# B&R Automation Studio project JOB_NUMBER (part 8)

### Device.var
```iecst
VAR
	Device : ARRAY[0..MAX_DEVICES] OF Device_typ := [(RequestRelease:=0,ReadyToRecieve:=0,Recieved:=0),221(0)];
END_VAR
VAR CONSTANT
	DEVICE_RELEASE_ID : UINT := 999; (**Value that is set in RequestRelease, when the destination is not required*)
	DEVICE_RELEASE_EMPTY : UINT := 998; (**Value that is set in RequestRelease, when the empty bag is required*)
	DEVICE_RECIEVE_WAIT : UINT := 997; (**Special ID to show a device is able to recieve but will not explicitly enable any sequence*)
END_VAR
```

### Device_IDS.var
```iecst
VAR CONSTANT
	MAX_DEVICES : UINT := 240;
END_VAR
(**Device ID constants*)
VAR CONSTANT
	DEVICE_LINE : ARRAY[0..99] OF UINT := [0,1,2,3,4,5,6,7,8,9,10,11,12,13,14,15,16,17,18,19,20,21,22,23,24,25,26,27,28,29,30,31,32,33,34,35,36,37,38,39,40,41,42,43,44,45,46,47,48,49,50,51,52,53,54,55,56,57,58,59,60,61,62,63,64,65,66,67,68,69,70,71,72,73,74,75,76,77,78,79,80,81,82,83,84,85,86,87,88,89,90,91,92,93,94,95,96,97,98,99]; (*Lines ID 1-99*)
	DEVICE_BSN : ARRAY[0..5] OF UINT := [0,101,102,103,104,105]; (*Bag Stacker Ongoing 101 - 105*)
	DEVICE_BSF : ARRAY[0..5] OF UINT := [0,106,107,108,109,110]; (*Bag Stacker Offgoing 106 - 110*)
	DEVICE_DC : ARRAY[0..10] OF UINT := [0,111,112,113,114,115,116,117,118,119,120]; (*Dischargers 111-120*)
	DEVICE_IC : ARRAY[0..10] OF UINT := [0,121,122,123,124,125,126,127,128,129,130]; (*Electric Inclines 121 - 130*)
	DEVICE_VC : ARRAY[0..10] OF UINT := [0,131,132,133,134,135,136,137,138,139,140]; (*VCs & Hoists 131 - 140*)
	DEVICE_TB : ARRAY[0..5] OF UINT := [0,141,142,143,144,145]; (*Transfer Belts 141 - 145*)
	DEVICE_PN : ARRAY[0..2] OF UINT := [0,146,147]; (*Ongoing Points 146 - 147*)
	DEVICE_PF : ARRAY[0..2] OF UINT := [0,148,149]; (*Points 148 - 149*)
	DEVICE_RPN : ARRAY[0..5] OF UINT := [0,151,152,153,154,155]; (*Rotary Ongoing 151-155*)
	DEVICE_RPF : ARRAY[0..5] OF UINT := [0,156,157,158,159,160]; (*Rotary Offgoing 156-160*)
	DEVICE_PC : ARRAY[0..10] OF UINT := [0,171,172,173,174,175,176,177,178,179,180]; (*Pneumatic VC 171-180*)
	DEVICE_PI : ARRAY[0..10] OF UINT := [0,181,182,183,184,185,186,187,188,189,190]; (*Pneumatic IC 181-190*)
	DEVICE_LU : ARRAY[0..10] OF UINT := [0,191,192,193,194,195,196,197,198,199,200]; (*Loading Units 191-200*)
	DEVICE_TRN : ARRAY[0..10] OF UINT := [0,201,202,203,204,205,206,207,208,209,210]; (*Twin Rail ongoing 201-205*)
	DEVICE_TRF : ARRAY[0..10] OF UINT := [0,211,212,213,214,215,216,217,218,219,220]; (*Twin Rail Offgoing 206-210*)
	DEVICE_POINT : ARRAY[0..20] OF UINT := [0,221,222,223,224,225,226,227,228,229,230,231,232,233,234,235,236,237,238,239,240]; (*Points 151 - 170*)
END_VAR
```

### Types.typ - Exported data types
```iecst
TYPE
	http_comm_typ : 	STRUCT
		Command : http_Cmd_typ; (**Set the values to pass into the http comm driver,*)
		Status : HTTP_Status_enum; (**Status of the http comm driver.*)
		LastError : STRING[60]; (**String to describe the last error*)
		lastResponse : httpResponseHeader_t;
		Overwrite : http_overwrite_t;
		ReplyCode : UINT; (**The response code *)
	END_STRUCT;
	http_Cmd_typ : 	STRUCT
		Method : UINT; (*Set the http cmd type.. POST,GET,PUT,DELETE*)
		Cmd_URL : dataPointer_typ; (*The string data appended to the URL - Use with GET and DELETE *)
		Body_Data : dataPointer_typ; (*Data to send in the body of the message - USE with POST and PUT*)
		ResponseData : dataPointer_typ; (*Data address of where to set the http response data*)
	END_STRUCT;
	dataPointer_typ : 	STRUCT
		Adr : UDINT;
		Size : UDINT;
	END_STRUCT;
	HTTP_Status_enum :
		(
		HTTP_COMM_STATUS_DISABLED,
		HTTP_COMM_STATUS_ACTIVE_WAIT_BUF,
		HTTP_COMM_STATUS_IN_BUFFER,
		HTTP_COMM_STATUS_IN_PROCESS,
		HTTP_COMM_STATUS_COMPLETE,
		HTTP_COMM_STATUS_ERROR
		);
	httpConfig_typ : 	STRUCT
		Host : STRING[20];
		Port : UINT;
	END_STRUCT;
	http_overwrite_t : 	STRUCT
		Host : BOOL; (**Set this to overwrite the host name and Port*)
		RequestHeader : BOOL; (**Set this to overwrite the Request Header*)
		Host_Config : httpConfig_typ; (**This data will overwrite the default host config*)
		RequestHeader_Data : httpRequestHeader_t; (**This data will overwrite the default request header.*)
	END_STRUCT;
END_TYPE
```

### Program Logical/Bag/http_Lib/httpServer (IEC, version 2.00.7) - *Listen for http requests

#### Variables.var - Local variables
```iecst
VAR
	httpServer : httpService;
	sendResponse : BOOL;
	abortResponse : BOOL;
	URI : STRING[500];
	requestHeader : httpRequestHeader_t;
	requestData : STRING[10000];
	responseHeader : httpResponseHeader_t;
	responseData : STRING[10000];
	Statistics : httpStatistics_t;
	serviceName : STRING[50];
	getParameterName : httpGetParameter;
END_VAR
VAR CONSTANT
	STRING_DOLLAR : STRING[1] := '&';
END_VAR
VAR
	activeFunction : UINT;
	mis : UDINT;
	bagIndex : UDINT;
	dst : USINT;
	error : INT;
	api : UINT;
	errorResponse : BOOL;
	overRideData : overRide_typ;
	ton_httpTimeOut : TON_10ms;
	recv : R_TRIG;
	wait : F_TRIG;
	cat : UDINT;
	cus : UDINT;
	bag : REFERENCE TO Bag_typ;
	prg : USINT;
	found : USINT;
	recieved : BOOL;
END_VAR
VAR CONSTANT
	BLANK_RESPONSE_HEADER : httpResponseHeader_t := (0);
END_VAR
VAR
	requestArriveTime : DATE_AND_TIME;
	debugCount : UDINT;
	index : UDINT;
	belt : USINT;
	velocity : INT;
(*	PartLoad : ARRAY[0..MAX_DISPLAYS] OF BOOL;*)
	direction : USINT;
	command : USINT;
END_VAR
```

#### Main.st - Init, cyclic, exit code
```iecst
//V2.00.1 -- TR. First release using version numbering
//V2.00.2 -- TR. Remove old http server functions FOR ABB settings as vars have been removed
//		  -- FIX: 200 OK could be returned in error
//V2.00.3 -- ADD: Load new configuration file command
//V2.00.4 -- REMOVE: Clear up old API Calls
//V2.00.5 -- Add Discharger Displays
//V2.00.6 -- ADD Part load and ABB Manual Controls (NEEDS ABB DRIVER 3.00.2)
//V2.00.7 -- ADD more functionality to ABB Manual Controls (Command and Direction) -- Also startup UDP Data connection
PROGRAM _INIT
	serviceName := 'supertrackPLC.api';
	httpServer.pServiceName := ADR(serviceName);
	httpServer.pUri := ADR(URI);
	httpServer.uriSize := SIZEOF(URI);
	httpServer.pRequestHeader := ADR(requestHeader);
	httpServer.pRequestData := ADR(requestData);
	httpServer.requestDataSize := SIZEOF(requestData);
	httpServer.pResponseHeader := ADR(responseHeader);
	httpServer.pResponseData := ADR(responseData);

	httpServer.pStatistics := ADR(Statistics);

	httpServer.option := httpOPTION_HTTP_11 + httpOPTION_SERVICE_TYPE_ROOT; //HTTP 1.1
	httpServer.enable := 0;

END_PROGRAM

PROGRAM _CYCLIC

	_httpServer;

	wait(CLK := (httpServer.phase = httpPHASE_SENDING));
	recv(CLK := (httpServer.phase = httpPHASE_RECEIVED));
	IF wait.Q THEN
		memset(ADR(responseData),0,SIZEOF(responseData));//Clear responseData
	END_IF;

	IF EDGEPOS(recieved) THEN
		requestArriveTime := CurrentTimestamp; // Get time stamp when the request arrives.
	END_IF;

	IF recieved THEN//recv.Q THEN
		//Get the API!
		api := FindAPI(URI,serviceName);

		CASE api OF

			API_UNKNOWN:
				errorResponse := 1;
				overRideData.responseHeader.status := '501 Not Implemented';
				responseData := 'Unknown API';
				httpServer.responseDataLen := LEN(responseData);

			API_MAINTENANCE_CONFIRM_REENTRY:
				sendResponse := 1;

			API_ST_FUNCTIONS://Legacy function => ?function=xxx
				_apiFunctions;

			API_CONFIG_LOAD_NEW: // Request to load new configuration.
				IF (Configuration.Interface.Status.LastLoaded >= requestArriveTime)  THEN // Send 200 OK when we see that the configuration is newer than the previous
					sendResponse := 1;
				ELSIF Configuration.Interface.Status.Error THEN
					errorResponse := 1;
					overRideData.responseHeader.status := '500 Internal Server Error';
					responseData := 'Failed to load file';
					httpServer.responseDataLen := LEN(responseData);
				ELSIF NOT Configuration.Interface.Cmd.Load AND (Configuration.Interface.Status.LastLoaded < requestArriveTime) THEN
					Configuration.Interface.Cmd.Load := 1;
					debugCount := debugCount + 1;
				END_IF;

			API_DISCHARGER_SUBMIT:

				getParameterName.searchString := requestData;
				getParameterName.searchOffset := 0;
				getParameterName.searchEndProperty := STRING_DOLLAR;
				//Find the first part of the array in JSON
				getParameterName.searchPropertyName := 'playId":"';
				getParameterName.searchEndProperty := '",';
				getParameterName();
				IF (getParameterName.status = ERR_OK) THEN
					index := DINT_TO_UDINT(atoi(ADR(getParameterName.outputValue)));
					IF (index <= MAX_DISPLAYS) THEN
						DischargerDisplaySubmit[index] := 1;
					END_IF;
					sendResponse := 1;
				ELSE
					errorResponse := 1;
					overRideData.responseHeader.status := '404 Not Found';
					responseData := 'Unknown display';
					httpServer.responseDataLen := LEN(responseData);
				END_IF;

			API_ABB_MANUAL_CMD:
				_abbManual;

			API_DATA_ENTRY_PARTLOAD:
				getParameterName.searchString := requestData;
				getParameterName.searchOffset := 0;
				getParameterName.searchEndProperty := STRING_DOLLAR;
				//Find the first part of the array in JSON
				getParameterName.searchPropertyName := 'playId":';
				getParameterName.searchEndProperty := '}';
				getParameterName();
				IF (getParameterName.status = ERR_OK) THEN
					index := DINT_TO_UDINT(atoi(ADR(getParameterName.outputValue)));
					IF (index <= MAX_DISPLAYS) THEN
						PartLoad[index] := 1;
					END_IF;
					sendResponse := 1;
				ELSE
					errorResponse := 1;
					overRideData.responseHeader.status := '404 Not Found';
					responseData := 'Unknown display';
					httpServer.responseDataLen := LEN(responseData);
				END_IF;

			//			API_CUSTOM_BELT_CONFIG:
			//				_setBeltConfig;
			//				sendResponse := 1;
			//
			//			API_CUSTOM_VC_COMMAND:
			//				_vcCommand;
			//
			//			API_LOADING_DATA:
			//				_getLoadingData;

		END_CASE;
	ELSE
		api := 0;
		activeFunction := 0;
	END_IF;

END_PROGRAM

PROGRAM _EXIT
	//Disable the Server on Exit..
	httpServer.enable := 0;
	httpServer();
END_PROGRAM
```

### ContactronTrip.var
```iecst
VAR CONSTANT
	CONTACTRON_TRIP_MIN : USINT := 2#00000001; (*Overload current must be set in % in 15 increments*)
	CONTACTRON_TRIP_50_PERCENT : USINT := 2#00000111;
	CONTACTRON_TRIP_MAX : USINT := 2#00001111;
END_VAR
```

### IOLink.var
```iecst
VAR
	IO_Link : IO_Link_Type;
	Fuse_PB_Reset : ARRAY[0..2] OF BOOL;
	Fuse_PB_Lamp : ARRAY[0..2] OF BOOL;
END_VAR
```

### Program Logical/IOLink/IOLink_Driver (IEC)

#### Main.st - Init, cyclic, exit code
```iecst
(********************************************************************
 * COPYRIGHT --
 ********************************************************************
 * PROGRAM: IOLink
 * File: IOLink_Driver.st
 * Author: Stephen Healey
 * Created: Sept 05, 2018
 ********************************************************************
 * Implementation OF PROGRAM IOLink
 ********************************************************************)
//V1.00.1 First Release

//	Description
//IOLink task for controlling Contactron's and EasyB's
//Constants need to be set. MAX_CONTACTRON and MAX_EASYB should match the hardware
//IO needs to be mapped for the Contactron's in the X20DS438A
//EasyB's IO does not need mapping. The interface still needs enabling in the X20DS438A config

//-------------------------------------------------------------
//-----------------------------Init----------------------------
//-------------------------------------------------------------
//	1.	Configures IOLink physical device, adjust address as needed
//	2.	Resets the controller state, needs to start offset, not 0

//-------------------------------------------------------------
//-----------------------------Cyclic--------------------------
//-------------------------------------------------------------
//	1.	Calls contactron action only if MAX_CONTACTRON is greater than zero
//	2.	Calls easyB action only if MAX_EASYB is greater than zero
//	3.	Monitors tripped status of all the EasyB's and enables reseting

//Use the following charts when setting the trip currents for the IOLink devices

//Contactron 												EasyB
//Current Setting Chart							Current Setting Chart
//Bit 		Nominal current						Enum										USINT			Value
//3 2 1 0 [mA]																													[mA]
//				 3 A 9 A
//0 0 0 0 180 1500									TRIP_CURRENT_DEFAULT		0					N/A
//0 0 0 1 300 2000									TRIP_CURRENT_500mA			5					500
//0 0 1 0 440 2500									TRIP_CURRENT_1A					10				1000
//0 0 1 1 600 3000									TRIP_CURRENT_2A					20				2000
//0 1 0 0 680 3500									TRIP_CURRENT_3A					30				3000
//0 1 0 1 880 4000									TRIP_CURRENT_4A					40				4000
//0 1 1 0 1000 4500									TRIP_CURRENT_5A					50				5000
//0 1 1 1 1100 5000									TRIP_CURRENT_6A					60				6000
//1 0 0 0 1200 5500									TRIP_CURRENT_8A					80				8000
//1 0 0 1 1500 6000									TRIP_CURRENT_10A				100				10000
//1 0 1 0 1600 6500
//1 0 1 1 1900 7000
//1 1 0 0 2100 7500
//1 1 0 1 2400 8000
//1 1 1 0 2700 8500
//1 1 1 1 3000 9000

PROGRAM _INIT
	//Configuration

	//Reset state

	backUp.fileDevice := 'UserPart';
	backUp.filePath := 'FuseTripConfig';

	//Load from file on boot

	backUp.step := backUpOpen;

	FOR n := 1 TO MAX_CONTACTRON DO
		IO_Link.Contactron[n].Cmd.Direction			:= CONTACTRON_FORWARD;
		IO_Link.Contactron[n].Cmd.Reset_Automatic	:= 1;
	END_FOR;

END_PROGRAM

PROGRAM _CYCLIC
	//Call status
	IF IO_Link.Status THEN
	 _status;
	END_IF;

	//Call httpResponse conditionally
//	IF IO_Link.Load THEN
//		_backUpRead;
//		_encodeData;
//	END_IF;

	//Call httpRequest conditionally
//	IF IO_Link.Save THEN
//		_decodeData;
//		_backUpWrite;
//		_encodeData;
//	END_IF;

	//Call contactron action
	IF MAX_CONTACTRON > 0 THEN
		_Contactron;
	END_IF;

//	//Call easy b action
//	IF (MAX_EASYB > 0) AND (MAX_EASYB <= 40) THEN
//		_EasyB;
//
//		//Monitor Tripped status
//		IO_Link.EasyB.Tripped := FALSE;
//		FOR n:=1 TO MAX_EASYB DO
//			IF IO_Link.EasyB.EasyB_Array[n].Status.TripState = EASYB_TRIPPED THEN
//				IO_Link.EasyB.Tripped := TRUE;
//				EXIT;
//			END_IF;
//		END_FOR;
//		//Reset Tripped status
//		IF IO_Link.EasyB.Tripped AND IO_Link.EasyB.Reset THEN
//			FOR n:=1 TO MAX_EASYB DO
//				IF IO_Link.EasyB.EasyB_Array[n].Status.TripState = EASYB_TRIPPED THEN
//					IO_Link.EasyB.EasyB_Array[n].Cmd.Reset := TRUE;
//				END_IF;
//			END_FOR;
//			IO_Link.EasyB.Reset := FALSE;
//		END_IF;
//		IO_Link.EasyB.TrippedLamp := IO_Link.EasyB.Tripped AND Std.Clock1s;
//	END_IF;

END_PROGRAM
```

#### _Contactron.st
```iecst
ACTION _Contactron:
	//----------------------------------------------
	//-----------------Contactron-------------------
	//----------------------------------------------

	//Write control word
	FOR n:=1 TO MAX_CONTACTRON DO
		IO_Link.Contactron[n].Comms.Read.CurrentActual := IO_Link.Contactron[n].Comms.Read.Data[0];
		IO_Link.Contactron[n].Comms.Read.DeviceType := IO_Link.Contactron[n].Comms.Read.Data[1];
		IO_Link.Contactron[n].Comms.Read.ThermalPercentOfMax := IO_Link.Contactron[n].Comms.Read.Data[2];
		IO_Link.Contactron[n].Comms.Read.CurrentPercentOfMax := IO_Link.Contactron[n].Comms.Read.Data[3];
		IO_Link.Contactron[n].Comms.Read.CurrentStatus := IO_Link.Contactron[n].Comms.Read.Data[4];
		IO_Link.Contactron[n].Comms.Read.Diagnostics := IO_Link.Contactron[n].Comms.Read.Data[5];

		CASE IO_Link.Contactron[n].Cmd.Direction OF
			CONTACTRON_FORWARD:
				IO_Link.Contactron[n].Comms.Write.Control.0 := IO_Link.Contactron[n].Cmd.Run;
				IO_Link.Contactron[n].Comms.Write.Control.7 := IO_Link.Contactron[n].Cmd.Run;
				IO_Link.Contactron[n].Comms.Write.Control.1 := FALSE;
				IO_Link.Contactron[n].Comms.Write.Control.5 := FALSE;

			CONTACTRON_REVERSE:
				IO_Link.Contactron[n].Comms.Write.Control.0 := FALSE;
				IO_Link.Contactron[n].Comms.Write.Control.7 := FALSE;
				IO_Link.Contactron[n].Comms.Write.Control.1 := IO_Link.Contactron[n].Cmd.Run;
				IO_Link.Contactron[n].Comms.Write.Control.5 := IO_Link.Contactron[n].Cmd.Run;

			ELSE
				IO_Link.Contactron[n].Comms.Write.Control.0 := FALSE;
				IO_Link.Contactron[n].Comms.Write.Control.7 := FALSE;
				IO_Link.Contactron[n].Comms.Write.Control.1 := FALSE;
				IO_Link.Contactron[n].Comms.Write.Control.5 := FALSE;

		END_CASE;

		IO_Link.Contactron[n].Comms.Write.Control.2 := IO_Link.Contactron[n].Cmd.Reset_Manual;
		IO_Link.Contactron[n].Comms.Write.Control.3 := IO_Link.Contactron[n].Cmd.Reset_Automatic;
		IO_Link.Contactron[n].Comms.Write.Control.4 := FALSE; //NOT USED
		IO_Link.Contactron[n].Comms.Write.Control.6 := IO_Link.Contactron[n].Cmd.Stop;

		IF IO_Link.Contactron[n].Cmd.Current > 0 THEN //Write trip current level
			IO_Link.Contactron[n].Comms.Write.NominalCurrent := (IO_Link.Contactron[n].Cmd.Current OR CONTACTRON_WRITE_CURRENT);
		ELSE
			IO_Link.Contactron[n].Comms.Write.NominalCurrent := 0;
		END_IF;
		IF IO_Link.Contactron[n].Cmd.Current = (IO_Link.Contactron[n].Comms.Read.CurrentStatus AND CONTACTRON_CURRENT_STATUS) THEN
			IO_Link.Contactron[n].Cmd.Current := 0; //Reset trip current if cmd written
		END_IF;

		//Read status
		IO_Link.Contactron[n].Status.Error := IO_Link.Contactron[n].Comms.Read.Diagnostics.0;
		IO_Link.Contactron[n].Status.STO_Active := NOT IO_Link.Contactron[n].Comms.Read.Diagnostics.3;
		IO_Link.Contactron[n].Status.Device_Ok := IO_Link.Contactron[n].Comms.Read.Diagnostics.5;
		IO_Link.Contactron[n].Status.Overload_Warning := IO_Link.Contactron[n].Comms.Read.Diagnostics.6;
		IO_Link.Contactron[n].Status.MainsFailure := ((IO_Link.Contactron[n].Comms.Read.CurrentStatus AND CONTACTRON_TRIP_STATUS) = CONTACTRON_MAINS_LOSS);
		IO_Link.Contactron[n].Status.PhaseLoss := ((IO_Link.Contactron[n].Comms.Read.CurrentStatus AND CONTACTRON_TRIP_STATUS) = CONTACTRON_PHASE_LOSS);
		IO_Link.Contactron[n].Status.Current := IO_Link.Contactron[n].Comms.Read.CurrentActual * 0.01;
		IO_Link.Contactron[n].Status.DeviceType := IO_Link.Contactron[n].Comms.Read.DeviceType;

		IF 	(IO_Link.Contactron[n].Comms.Read.CurrentStatus = 0) THEN
			IO_Link.Contactron[n].Cmd.Current				:= CONTACTRON_TRIP_50_PERCENT;
		END_IF;

	END_FOR;
END_ACTION
```

### Program Logical/IOLink/FuseManagement (IEC, version 1.00.2)

#### Main.st - Init, cyclic, exit code
```iecst
//V1.00.0 -- First Release
//V1.00.1 -- Update so we monitor the status of the fuse and can send reset commands
//V1.00.2 -- Invert the fault lamp to a healthy lamp to stay consistent with hardwired devices

PROGRAM _INIT
Fuse[1].pDevice := ADR('SL1.IF1.ST11.IF1.ST8.IF1');//'SL1.IF1.ST2.IF1.ST7.IF1');
Fuse[2].pDevice := ADR('SL1.IF1.ST11.IF1.ST8.IF2');
Fuse[3].pDevice := ADR('SL1.IF1.ST11.IF1.ST8.IF3');
Fuse[4].pDevice := ADR('SL1.IF1.ST11.IF1.ST8.IF4');
Fuse[5].pDevice := ADR('SL1.IF1.ST21.IF1.ST8.IF1');
Fuse[6].pDevice := ADR('SL1.IF1.ST21.IF1.ST8.IF2');
Fuse[7].pDevice := ADR('SL1.IF1.ST21.IF1.ST8.IF3');
Fuse[8].pDevice := ADR('SL1.IF1.ST21.IF1.ST8.IF4');

FOR n := 1 TO MAX_FUSE_BANKS DO
	fuse ACCESS ADR(Fuse[n]);
	fuse.Write.MinVoltage := 1800;
	fuse.Write.MaxVoltage := 2800;
	FOR i := 1 TO MAX_FUSES DO
		fuse.Write.Channel[i].Status := EB_STATE_ON;
		fuse.Write.Channel[i].TripCurrent := 40;
	END_FOR;
	fuse.index := 90;
	fuse.readStatusOnly := 0;
	fuseTrippedAlarm[n] := 0;
END_FOR;

//alarm 	ACCESS ADR(Alarm[208]);
END_PROGRAM

PROGRAM _CYCLIC

IF EDGEPOS(X[1003].X04) THEN
	reset[0] := 1;
END_IF;
IF EDGEPOS(X[2003].X04) THEN
	reset[1] := 1;
END_IF;

fuseFault[0] := 0;
fuseFault[1] := 0;
//alarm.On	:= 0;
//alarm.Name	:= 0;

FOR n := 1 TO MAX_FUSE_BANKS DO
	fuse ACCESS ADR(Fuse[n]);
	read ACCESS ADR(fuse.IOLinkRead);
	write ACCESS ADR(fuse.IOLinkWrite);

	read.enable := 1;
	write.enable := 1;
	write.pDeviceName 	:= fuse.pDevice;
	read.pDeviceName 	:= fuse.pDevice;

	IF EDGEPOS(read.readLen > 0) THEN
		count := count + 1;
	END_IF;

	IF (read.errorCode > 0) THEN
		fuse.index := 10;
	END_IF;

	IF (n < 5) THEN
		plc := 0;
	ELSE
		plc := 1;
	END_IF;

	CASE fuse.index	OF
		0:

		32:	//Read Error Count
			read.datatype 		:= ioLinkTYPE_SINT;
			read.pData			:= ADR(fuse.Read.ErrorCount);
			read.dataLen		:= SIZEOF(fuse.Read.ErrorCount);
			read.index			:= fuse.index;
			read.subIndex		:= 0;
			read();
			IF read.status = ERR_OK THEN
				fuse.index := fuse.index + 1;
			ELSIF (read.status <> ERR_FUB_BUSY) AND (read.status <> ERR_FUB_ENABLE_FALSE)  THEN
				fuse.index := fuse.index + 1;
				//fuse.Read.ErrorCount := 0;
			END_IF;

		33://
			fuse.index := 36;

		36://Device Status	 R/O USINT
			read.datatype 		:= ioLinkTYPE_SINT;
			read.pData			:= ADR(fuse.Read.DeviceStatus);
			read.dataLen		:= SIZEOF(fuse.Read.DeviceStatus);
			read.index			:= fuse.index;
			read.subIndex		:= 0;
			read();
			IF read.status = ERR_OK THEN
				fuse.index := fuse.index + 1;
			ELSIF (read.status <> ERR_FUB_BUSY) AND (read.status <> ERR_FUB_ENABLE_FALSE)  THEN
				fuse.index := fuse.index + 1;
				//fuse.Read.ErrorCount := 0;
			END_IF;

		37:// Device Status	 R/O String
			read.datatype 		:= ioLinkTYPE_STRING;
			read.pData			:= ADR(fuse.Read.DeviceStatusString);
			read.dataLen		:= SIZEOF(fuse.Read.DeviceStatusString);
			read.index			:= fuse.index;
			read.subIndex		:= 0;
			read();
			IF read.status = ERR_OK THEN
				fuse.index := fuse.index + 1;
			ELSIF (read.status <> ERR_FUB_BUSY) AND (read.status <> ERR_FUB_ENABLE_FALSE)  THEN
				fuse.index := fuse.index + 1;
				//fuse.Read.ErrorCount := 0;
			END_IF;

		38:
			fuse.index := 80;

		80://
			IF (fuse.trip > 0) THEN
				command := UINT_TO_USINT((fuse.trip * 5) - 2); // <--RESET //((fuse.trip * 5) - 4); //<-- ON

				write.datatype 		:= ioLinkTYPE_USINT;
				write.pData			:= ADR(command);
				write.dataLen		:= SIZEOF(command);
				write.index			:= fuse.index;
				write.subIndex		:= 0;
				write();
				IF (write.status = ERR_OK) THEN
					fuse.index := fuse.index + 1;	;
				ELSIF (write.status <> ERR_FUB_BUSY) AND (write.status <> ERR_FUB_ENABLE_FALSE) THEN
					fuse.index := fuse.index + 1;
				END_IF;
			ELSE
				fuse.index := fuse.index + 1;
			END_IF;

		81://Gateway options ? R/W
			IF fuse.Write.AutoNodeAllocation_Off OR fuse.Write.AutoNodeAllocation_On  THEN
				//1 is automatic allocation off!
				//0 is on?
				IF fuse.Write.AutoNodeAllocation_Off THEN
					write.datatype 		:= ioLinkTYPE_RECORD;
					gatewayOption 		:= 1;
					write.subIndex		:= 1;
				ELSE
					write.datatype 		:= ioLinkTYPE_SINT;
					gatewayOption 		:= 0;
					write.subIndex		:= 0 ;
				END_IF;
				write.pData			:= ADR(gatewayOption);
				write.dataLen		:= 1;
				write.index			:= fuse.index;
				write();
				IF (write.status = ERR_OK) THEN
					fuse.index := fuse.index + 1;	;
					fuse.Write.AutoNodeAllocation_On := 0;
					fuse.Write.AutoNodeAllocation_Off := 0;
				ELSIF (write.status <> ERR_FUB_BUSY) AND (write.status <> ERR_FUB_ENABLE_FALSE) THEN
					fuse.index := fuse.index + 1;
					fuse.Write.AutoNodeAllocation_On := 0;
					fuse.Write.AutoNodeAllocation_Off := 0;
				END_IF;

			ELSE // Read if no write
				read.datatype 		:= ioLinkTYPE_SINT;
				read.pData			:= ADR(fuse.Read.GatewayOptions);
				read.dataLen		:= SIZEOF(fuse.Read.GatewayOptions);
				read.index			:= fuse.index;
				read.subIndex		:= 0;
				read();
				IF read.status = ERR_OK THEN
					fuse.index := fuse.index + 1;
				ELSIF (read.status <> ERR_FUB_BUSY) AND (read.status <> ERR_FUB_ENABLE_FALSE)  THEN
					fuse.index := fuse.index + 1;
				END_IF;
			END_IF;

		82://Set breaker 1 options to all
			fuse.index := 90;

		83:// Reset individual breaker.

		90://Input Voltage
			read.datatype 		:= ioLinkTYPE_INT;
			read.pData			:= ADR(fuse.Read.InputVoltage);
			read.dataLen		:= SIZEOF(fuse.Read.InputVoltage);
			read.index			:= fuse.index;
			read.subIndex		:= 0;
			read();
			IF read.status = ERR_OK THEN
				fuse.index := fuse.index + 1;
			ELSIF (read.status <> ERR_FUB_BUSY) AND (read.status <> ERR_FUB_ENABLE_FALSE)  THEN
				fuse.index := fuse.index + 1;
			END_IF;

		91://Number of Nodes
			read.datatype 		:= ioLinkTYPE_USINT;
			read.pData			:= ADR(fuse.Read.NoNodes);
			read.dataLen		:= SIZEOF(fuse.Read.NoNodes);
			read.index			:= fuse.index;
			read.subIndex		:= 0;
			read();
			IF read.status = ERR_OK THEN
				IF (fuse.Read.NoNodes > MAX_FUSES) THEN
					fuse.Read.NoNodes := MAX_FUSES;
				END_IF;
				fuse.index := fuse.index + 1;
			ELSIF (read.status <> ERR_FUB_BUSY) AND (read.status <> ERR_FUB_ENABLE_FALSE)  THEN
				fuse.Read.NoNodes := 0;
				fuse.index := fuse.index + 1;
			END_IF;

		92://
			fuse.index := 100;

		100:// Max Voltage
			IF (fuse.Write.MaxVoltage > 0) THEN

				write.datatype 		:= ioLinkTYPE_INT;
				write.pData			:= ADR(fuse.Write.MaxVoltage);
				write.dataLen		:= SIZEOF(fuse.Write.MaxVoltage);
				write.index			:= fuse.index;
				write.subIndex		:= 0;
				write();
				IF (write.status = ERR_OK) THEN
					fuse.index := fuse.index + 1;
					fuse.Read.MaxVoltage := fuse.Write.MaxVoltage;
					fuse.Write.MaxVoltage := 0;
				ELSIF (write.status <> ERR_FUB_BUSY) AND (write.status <> ERR_FUB_ENABLE_FALSE) THEN
					fuse.index := fuse.index + 1;
					fuse.Write.MaxVoltage := 0;
				END_IF;
			ELSE // Read if no write

				read.datatype 		:= ioLinkTYPE_INT;
				read.pData			:= ADR(fuse.Read.MaxVoltage);
				read.dataLen		:= SIZEOF(fuse.Read.MaxVoltage);
				read.index			:= fuse.index;
				read.subIndex		:= 0;
				read();
				IF read.status = ERR_OK THEN
					fuse.index := fuse.index + 1;
				ELSIF (read.status <> ERR_FUB_BUSY) AND (read.status <> ERR_FUB_ENABLE_FALSE)  THEN
					fuse.index := fuse.index + 1;
					fuse.Read.MaxVoltage := 0;
				END_IF;
			END_IF;

		101://MinVoltage
			IF (fuse.Write.MinVoltage > 0) THEN
				write.datatype 		:= ioLinkTYPE_INT;
				write.pData			:= ADR(fuse.Write.MinVoltage);
				write.dataLen		:= SIZEOF(fuse.Write.MinVoltage);
				write.index			:= fuse.index;
				write.subIndex		:= 0;
				write();
				IF (write.status = ERR_OK) THEN
					fuse.index := fuse.index + 1;
					fuse.Read.MinVoltage :=	fuse.Write.MinVoltage;
					fuse.Write.MinVoltage := 0;
				ELSIF (write.status <> ERR_FUB_BUSY) AND (write.status <> ERR_FUB_ENABLE_FALSE) THEN
					fuse.index := fuse.index + 1;
					fuse.Write.MinVoltage := 0;
				END_IF;
			ELSE // Read if no write

				read.datatype 		:= ioLinkTYPE_INT;
				read.pData			:= ADR(fuse.Read.MinVoltage);
				read.dataLen		:= SIZEOF(fuse.Read.MinVoltage);
				read.index			:= fuse.index;
				read.subIndex		:= 0;
				read();
				IF read.status = ERR_OK THEN
					fuse.index := fuse.index + 1;
				ELSIF (read.status <> ERR_FUB_BUSY) AND (read.status <> ERR_FUB_ENABLE_FALSE)  THEN
					fuse.index := fuse.index + 1;
					fuse.Read.MinVoltage := 0;
				END_IF;
			END_IF;

		102:// Enable Events R/W
			IF (fuse.Write.EnableEvents > 0) THEN
				write.datatype 		:= ioLinkTYPE_SINT;
				write.pData			:= ADR(fuse.Write.EnableEvents);
				write.dataLen		:= SIZEOF(fuse.Write.EnableEvents);
				write.index			:= fuse.index;
				write.subIndex		:= 0;
				write();
				IF (write.status = ERR_OK) THEN
					fuse.index := fuse.index + 1;
					fuse.Write.EnableEvents := 0;
				ELSIF (write.status <> ERR_FUB_BUSY) AND (write.status <> ERR_FUB_ENABLE_FALSE) THEN
					fuse.index := fuse.index + 1;
					fuse.Write.EnableEvents := 0;
				END_IF;
			ELSE // Read if no write

				read.datatype 		:= ioLinkTYPE_SINT;
				read.pData			:= ADR(fuse.Read.EnableEvents);
				read.dataLen		:= SIZEOF(fuse.Read.EnableEvents);
				read.index			:= fuse.index;
				read.subIndex		:= 0;
				read();
				IF read.status = ERR_OK THEN
					fuse.index := fuse.index + 1;
				ELSIF (read.status <> ERR_FUB_BUSY) AND (read.status <> ERR_FUB_ENABLE_FALSE)  THEN
					fuse.index := fuse.index + 1;
					fuse.Read.EnableEvents := 0;
				END_IF;
			END_IF;

		103:
			fuse.index := 201;

		201..240://Read Only Trip Counter
			index := (fuse.index - 200);
			read.datatype 		:= ioLinkTYPE_SINT;
			read.pData			:= ADR(fuse.Read.Channel[index].TripCount);
			read.dataLen		:= SIZEOF(fuse.Read.Channel[index].TripCount);
			read.index			:= fuse.index;
			read.subIndex		:= 0;
			read();
			IF read.status = ERR_OK THEN
				fuse.index := fuse.index + 1;
			ELSIF (read.status <> ERR_FUB_BUSY) AND (read.status <> ERR_FUB_ENABLE_FALSE)  THEN
				fuse.index := fuse.index + 1;
				//fuse.Read.Channel[index].TripCount := 0;
			END_IF;

		241:
			fuse.index := 301;

		301..340://Read only Actaul Current
			index := (fuse.index - 300);
			read.datatype 		:= ioLinkTYPE_INT;
			read.pData			:= ADR(fuse.Read.Channel[index].ActCurrent);
			read.dataLen		:= SIZEOF(fuse.Read.Channel[index].ActCurrent);
			read.index			:= fuse.index;
			read.subIndex		:= 0;
			read();
			IF read.status = ERR_OK THEN
				IF (fuse.index < (300 + fuse.Read.NoNodes)) THEN
					fuse.index := fuse.index + 1;
				ELSE
					fuse.index := 401;
				END_IF;
			ELSIF (read.status <> ERR_FUB_BUSY) AND (read.status <> ERR_FUB_ENABLE_FALSE)  THEN
				IF (fuse.index < (300 + fuse.Read.NoNodes)) THEN
					fuse.index := fuse.index + 1;
				ELSE
					fuse.index := 401;
				END_IF;
			END_IF;

		341:
			fuse.index := 401;

		401..440://Over Current
			index := (fuse.index - 400);
			IF (fuse.Write.Channel[index].TripCurrent > 0) THEN
				write.datatype 		:= ioLinkTYPE_SINT;
				write.pData			:= ADR(fuse.Write.Channel[index].TripCurrent);
				write.dataLen		:= SIZEOF(fuse.Write.Channel[index].TripCurrent);
				write.index			:= fuse.index;
				write.subIndex		:= 0;
				write();
				IF (write.status = ERR_OK) THEN
					IF (fuse.index < (400 + fuse.Read.NoNodes)) THEN
						fuse.index := fuse.index + 1;
					ELSE
						fuse.index := 441;
					END_IF;
					fuse.Read.Channel[index].TripCurrent := fuse.Write.Channel[index].TripCurrent;
					fuse.Write.Channel[index].TripCurrent := 0;
				ELSIF (write.status <> ERR_FUB_BUSY) AND (write.status <> ERR_FUB_ENABLE_FALSE) THEN
					IF (fuse.index < (400 + fuse.Read.NoNodes)) THEN
						fuse.index := fuse.index + 1;
					ELSE
						fuse.index := 441;
					END_IF;
					fuse.Write.Channel[index].TripCurrent := 0;
				END_IF;
			ELSE // Read if no write

				read.datatype 		:= ioLinkTYPE_USINT;
				read.pData			:= ADR(fuse.Read.Channel[index].TripCurrent);
				read.dataLen		:= SIZEOF(fuse.Read.Channel[index].TripCurrent);
				read.index			:= fuse.index;
				read.subIndex		:= 0;
				read();
				IF read.status = ERR_OK THEN
					IF (fuse.index < (400 + fuse.Read.NoNodes)) THEN
						fuse.index := fuse.index + 1;
					ELSE
						fuse.index := 441;
					END_IF;
				ELSIF (read.status <> ERR_FUB_BUSY) AND (read.status <> ERR_FUB_ENABLE_FALSE)  THEN
					IF (fuse.index < (400 + fuse.Read.NoNodes)) THEN
						fuse.index := fuse.index + 1;
					ELSE
						fuse.index := 441;
					END_IF;
					fuse.Read.Channel[index].TripCurrent := 0;
				END_IF;
			END_IF;

		441..500:
			fuse.index := 501;
			fuse.trip := 0;

		501..540://	status RO
			index := (fuse.index - 500);

			read.datatype 		:= ioLinkTYPE_USINT;
			read.pData			:= ADR(fuse.Read.Channel[index].Status);
			read.dataLen		:= SIZEOF(fuse.Read.Channel[index].Status);
			read.index			:= fuse.index;
			read.subIndex		:= 0;
			read();
			IF read.status = ERR_OK THEN
				IF (fuse.index < (500 + fuse.Read.NoNodes)) THEN
					fuse.index := fuse.index + 1;
				ELSE
					fuse.index := 541;
				END_IF;
			ELSIF (read.status <> ERR_FUB_BUSY) AND (read.status <> ERR_FUB_ENABLE_FALSE)  THEN
				IF (fuse.index < (500 + fuse.Read.NoNodes)) THEN

					CASE fuse.Read.Channel[index].Status OF
						EB_STATE_NC:

						EB_STATE_OFF:

						EB_STATE_ON:

						EB_STATE_TRIP:
							fuse.trip := index;
						EB_STATE_I_90:

						EB_STATE_I_100:

						EB_STATE_TRIP_HARDWARE:

						EB_STATE_TRIP_THERMAL:
							fuse.trip := index;

						EB_STATE_TRIP_SW_OFF:

					END_CASE;

					fuse.index := fuse.index + 1;
				ELSE
					fuse.index := 541;
				END_IF;
				fuse.Read.Channel[index].Status := 0;
			END_IF;

		541:
			IF reset[plc] THEN
				fuse.index := 80;
			ELSIF fuse.readStatusOnly THEN
				fuse.index := 500;
			ELSE
				fuse.index := 901;
			END_IF;
			IF (fuse.trip > 0) THEN
				fuseTrippedAlarm[n] := 1;
			ELSE
				fuseTrippedAlarm[n] := 0;
			END_IF;

		701..740://Options

		901..940:
			index := (fuse.index - 900);
			read.datatype 		:= ioLinkTYPE_USINT;
			read.pData			:= ADR(fuse.Read.Channel[index].Type);
			read.dataLen		:= SIZEOF(fuse.Read.Channel[index].Type);
			read.index			:= fuse.index;
			read.subIndex		:= 0;
			read();
			IF read.status = ERR_OK THEN
				IF (fuse.index < (900 + fuse.Read.NoNodes)) THEN
					fuse.index := fuse.index + 1;
				ELSE
					fuse.index := 941;
				END_IF;
			ELSIF (read.status <> ERR_FUB_BUSY) AND (read.status <> ERR_FUB_ENABLE_FALSE)  THEN
				IF (fuse.index < (900 + fuse.Read.NoNodes)) THEN
					fuse.index := fuse.index + 1;
				ELSE
					fuse.index := 941;
				END_IF;
				//fuse.Read.Channel[index].ActCurrent := 0;
			END_IF;

		941:
			fuse.index := 501;
			fuse.readStatusOnly := 1;

		998:// Test Write
			write.pData := ADR(testData);
			write();
			IF (write.status = ERR_OK) THEN
				fuse.index := 1000;
			ELSIF (write.status <> ERR_FUB_BUSY) AND (write.status <> ERR_FUB_ENABLE_FALSE) THEN
				fuse.index := 1001;
			END_IF;
		999:// Test Read
			read();
			IF (read.status = ERR_OK) THEN
				fuse.index := 1000;
			ELSIF (read.status <> ERR_FUB_BUSY) AND (read.status <> ERR_FUB_ENABLE_FALSE)  THEN
				fuse.index := 1001;
			END_IF;
		1000:// Test result

	END_CASE;

	IF fuseTrippedAlarm[n] THEN
		fuseFault[plc]	:= 1;
		//alarm.On	:= TRUE;
		//alarm.Name	:= ALM_FUSE_TRIPPED;
	END_IF;

	IF NOT fuseFault[plc] THEN
		reset[plc] := 0;
	END_IF;

END_FOR;

Y[1004].Y02 := NOT fuseFault[0];
Y[2004].Y02 := NOT fuseFault[1];

END_PROGRAM
```

#### Types.typ - Local data types
```iecst
(*Insert your comment here.*)

TYPE
	Fuse_typ : 	STRUCT
		pDevice : UDINT; (**pointer to Address on IO Link interface*)
		ProcessData : ARRAY[0..5]OF USINT;
		index : UINT; (**Setting Index*)
		Read : FuseRead_typ;
		Write : FuseWrite_typ;
		IOLinkRead : ioLinkRead;
		IOLinkWrite : ioLinkWrite;
		trip : UINT; (**We have detected a trip error*)
		readStatusOnly : BOOL; (**Bit to say all config params have been read- only cycle through the status to see if we have an error*)
	END_STRUCT;
	FuseWrite_typ : 	STRUCT
		MinVoltage : INT;
		MaxVoltage : INT;
		EnableEvents : USINT;
		AutoNodeAllocation_Off : BOOL;
		AutoNodeAllocation_On : BOOL;
		Channel : ARRAY[1..MAX_FUSES]OF FuseChannel_typ;
	END_STRUCT;
	FuseRead_typ : 	STRUCT
		MinVoltage : INT;
		MaxVoltage : INT;
		ErrorCount : UINT;
		Channel : ARRAY[1..MAX_FUSES]OF FuseChannel_Read_typ;
		DeviceStatus : USINT;
		DeviceStatusString : STRING[80];
		InputVoltage : UINT;
		NoNodes : USINT;
		EnableEvents : USINT;
		GatewayOptions : FuseGateway_enum;
	END_STRUCT;
	FuseGateway_enum :
		(
		EB_AUTO_NODE_OFF,
		EB_AUTO_NODE_ON
		);
	FuseType_enum :
		(
		EB_UNKNOWN := 0,
		EB_3824_100_0 := 170,
		EB_0824_100_0 := 138,
		EB_1824_010_0 := 145,
		EB_1824_020_0 := 146,
		EB_1824_030_0 := 147,
		EB_1824_040_0 := 148,
		EB_1824_060_0 := 150,
		EB_1824_080_0 := 152,
		EB_1824_100_0 := 154
		);
	FuseChannel_Read_typ : 	STRUCT
		TripCurrent : USINT; (*400 + Fuse Number*)
		Status : USINT;
		TripCount : SINT;
		ActCurrent : UINT;
		Type : FuseType_enum;
	END_STRUCT;
	FuseChannel_typ : 	STRUCT
		TripCurrent : USINT; (*400 + Fuse Number*)
		Status : USINT;
	END_STRUCT;
END_TYPE
```

#### Variables.var - Local variables
```iecst
VAR
	lastIndex : UINT;
	fuseTrippedAlarm : ARRAY[0..MAX_FUSE_BANKS] OF BOOL; (*alarm : REFERENCE TO Alm;*)
	i : USINT;
	testData : INT;
	gatewayOption : BOOL;
	count : UDINT;
	command : USINT;
	reset : ARRAY[0..2] OF BOOL;
	fuseFault : ARRAY[0..2] OF BOOL;
	read : REFERENCE TO ioLinkRead;
	write : REFERENCE TO ioLinkWrite;
	fuse : REFERENCE TO Fuse_typ;
	n : INT;
	Fuse : ARRAY[0..MAX_FUSE_BANKS] OF Fuse_typ;
	index : UINT;
END_VAR
VAR CONSTANT
	MAX_FUSE_BANKS : USINT := 8;
	MAX_FUSES : USINT := 40; (** Don;t set less than 40 the code will read the correct number*)
END_VAR
VAR
	plc : USINT;
END_VAR
```

### Library Logical/IOLink/IOLinkLib (IEC)
Depends on: AsIOLink

#### Constants.var - Exported constants
```iecst
VAR CONSTANT
	EASYB_STATE_5 : USINT := 5;
	EASYB_TRIPPED : USINT := 3;
	EASYB_SWITCHED_ON : USINT := 2;
	CONTACTRON_CURRENT_STATUS : USINT := 15;
	CONTACTRON_WRITE_CURRENT : USINT := 128;
	CONTACTRON_TRIP_STATUS : USINT := 112;
	CONTACTRON_MAINS_LOSS : USINT := 32;
	CONTACTRON_PHASE_LOSS : USINT := 64;
	MAX_CONTACTRON : USINT := 2;
END_VAR
```

### Program Logical/Programs/ModMaster

#### ModMaster.var
```iecst
(*-----------------------------------------------------------------------------------------------------------------------------------------------------------------------------------------------------------------------------------------*)
(*Modbus master function block and configuration*)
VAR
	ModbusTcpMaster : MBmaster;
	MasterConfig : modbus_master_cfg_typ := (0);
	reset_error : BOOL := FALSE;
END_VAR
(*IO sample arrays*)
VAR
	A_Out : ARRAY[0..20] OF UINT := [21(0)];
	A_In : ARRAY[0..20] OF UINT := [21(0)];
	D_Out : ARRAY[0..49] OF BOOL := [50(FALSE)];
	D_In : ARRAY[0..49] OF BOOL := [50(FALSE)];
END_VAR
(*MISC variables*)
VAR
	ip : STRING[20];
	logger : ARRAY[0..19] OF STRING[50];
	StartStop : BOOL := FALSE;
END_VAR
```

#### ModMaster.st
```iecst
(********************************************************************
 * COPYRIGHT --
 ********************************************************************
 * PROGRAM: ModMaster
 ********************************************************************
 * Implementation OF PROGRAM ModMaster
 ********************************************************************)

PROGRAM _INIT
	strcpy(ADR(ip), ADR('192.168.5.114'));					 (* Slave device IP address *)

	(* --------------------------------------------------------------------
	  Reset FUNCTION blocks AND data structure on startup (SGC)
	  --------------------------------------------------------------------- *)
    memset(ADR(ModbusTcpMaster), 0, SIZEOF(ModbusTcpMaster));
    memset(ADR(MasterConfig), 0, SIZEOF(MasterConfig));
    memset(ADR(logger), 0, SIZEOF(logger));

	(* --------------------------------------------------------------------
	  Sample FOR reading/writing data from/TO a modbusTCP slave
	  --------------------------------------------------------------------- *)
	MasterConfig.action_enable[0].cyclic 	:= 1;			(* Read data cyclic *)
	MasterConfig.action_param[0].p_pv		:= ADR(D_In);	(* Store data in this variable *)
	MasterConfig.action_param[0].quantity 	:= 6;			(* Number of items to read *)
	MasterConfig.action_param[0].unit 		:= 1;			(* Unit address - ignore if not specified *)
	MasterConfig.action_param[0].start_addr := 16#1F3C;		(* Read from this modbus address *)
	MasterConfig.action_param[0].timer 		:= 500;			(* Refresh timer for this item *)
	MasterConfig.action_param[0].type 		:= 2;			(* Function code for this item (2 := read discrete inputs) *)

	MasterConfig.action_enable[1].cyclic 	:= 1;			(* Write data cyclic *)
	MasterConfig.action_param[1].p_pv		:= ADR(D_Out); 	(* Take data from this address *)
	MasterConfig.action_param[1].quantity 	:= 2; 			(* Number of items to write *)
	MasterConfig.action_param[1].unit 		:= 1;			(* Unit address - ignore if not specified *)
	MasterConfig.action_param[1].start_addr := 16#1F42;		(* Write to this modbus address *)
	MasterConfig.action_param[1].timer 		:= 500; 		(* Refresh timer for this item *)
	MasterConfig.action_param[1].type 		:= 15; 			(* Function code for this item (15 := write multiple coils) *)

	MasterConfig.action_enable[2].cyclic 	:= 1; 			(* Read data cyclic *)
	MasterConfig.action_param[2].p_pv		:= ADR(A_In); 	(* Store data in this variable *)
	MasterConfig.action_param[2].quantity 	:= 6; 			(* Number of items to read *)
	MasterConfig.action_param[2].unit 		:= 1;			(* Unit address - ignore if not specified *)
	MasterConfig.action_param[2].start_addr := 7996; 		(* Read from this modbus address *)
	MasterConfig.action_param[2].timer 		:= 60; 		(* Refresh timer for this item *)
	MasterConfig.action_param[2].type 		:= 4; 			(* Function code for this item (4 := read inputs) *)

	MasterConfig.action_enable[3].cyclic 	:= 1; 			(* Write data cyclic *)
	MasterConfig.action_param[3].p_pv		:= ADR(A_Out); 	(* Take data from this address *)
	MasterConfig.action_param[3].quantity 	:= 2; 			(* Number of items to write *)
	MasterConfig.action_param[3].unit 		:= 1;			(* Unit address - ignore if not specified *)
	MasterConfig.action_param[3].start_addr := 8002; 		(* Write to this modbus address *)
	MasterConfig.action_param[3].timer 		:= 60; 		(* Refresh timer for this item *)
	MasterConfig.action_param[3].type 		:= 16; 			(* Function code for this item (16 := write holding register) *)

	(* --------------------------------------------------------------------
	  Sample FOR reading data from a modbusTCP slave
	  --------------------------------------------------------------------- *)
	ModbusTcpMaster.enable 			:= 1;						(* Start master *)
	ModbusTcpMaster.device			:= ADR('IF2'); 				(* Ethernet device string *)
	ModbusTcpMaster.slave_ip_addr 	:= ip; 						(* Transfer slave device IP address *)
	ModbusTcpMaster.p_cfg 			:= ADR(MasterConfig); 		(* Pointer to configuration *)
	ModbusTcpMaster.cycle_time 		:= 10; 						(* Master cycle time in ms *)

	(* The LOG information will show communication details. Enable for debugging,
	  disable FOR production TO save system resources *)
	ModbusTcpMaster.log.data_lines := 20; 						(* Number of logging lines *)
	ModbusTcpMaster.log.pData := ADR(logger); 					(* Pointer to logger string array *)
(*	StartStop := 1;*)
END_PROGRAM

PROGRAM _CYCLIC
	(* --------------------------------------------------------------------
	  Cyclic FUNCTION call
	  --------------------------------------------------------------------- *)
	IF(StartStop) THEN
		ModbusTcpMaster();
	END_IF

	(* --------------------------------------------------------------------
	  Reset last error information
	  --------------------------------------------------------------------- *)
	IF(reset_error) THEN
		memset(ADR(ModbusTcpMaster.last_error), 0, 2);
		reset_error := 0;
	END_IF
END_PROGRAM
```

### Program Logical/Programs/ModSlave

#### ModSlave.var
```iecst
(*-----------------------------------------------------------------------------------------------------------------------------------------------------------------------------------------------------------------------------------------*)
(*Modbus slave function block and configuration*)
VAR
	ModbusTcpSlave : MBslave := (0);
	SlaveConfig : modbus_slave_cfg_typ := (0);
	reset_error : BOOL := FALSE;
END_VAR
(*IO sample arrays*)
VAR
	DO_Bool : ARRAY[0..99] OF BOOL := [100(FALSE)];
	DI_Bool : ARRAY[0..99] OF BOOL := [100(FALSE)];
	AO_Word : ARRAY[0..99] OF UINT := [100(0)];
	AI_Word : ARRAY[0..99] OF UINT := [100(0)];
END_VAR
(*MISC variables*)
VAR
	idx : UINT := 0;
	logger : ARRAY[0..19] OF STRING[50] := [20(' ')];
	StartStop : BOOL := FALSE;
END_VAR
```

#### ModSlave.st
```iecst
(********************************************************************
 * COPYRIGHT --
 ********************************************************************
 * PROGRAM: ModSlave
 ********************************************************************
 * Implementation OF PROGRAM ModSlave
 ********************************************************************)

PROGRAM _INIT
	(* --------------------------------------------------------------------
	  Reset FUNCTION blocks AND data structure on startup (SGC)
	  --------------------------------------------------------------------- *)
    memset(ADR(ModbusTcpSlave), 0, SIZEOF(ModbusTcpSlave));
    memset(ADR(SlaveConfig), 0, SIZEOF(SlaveConfig));
    memset(ADR(logger), 0, SIZEOF(logger));

	(* --------------------------------------------------------------------
	  Create default IO mapping FOR digital AND analog area
	  --------------------------------------------------------------------- *)
	FOR idx:=0 TO SIZEOF(DO_Bool)-1 DO
		SlaveConfig.p_coils[idx] := ADR(DO_Bool[idx]);
	END_FOR;
	FOR idx:=0 TO SIZEOF(DI_Bool)-1 DO
		SlaveConfig.p_discrete_inputs[idx]	:= ADR(DI_Bool[idx]);
	END_FOR;
	FOR idx:=0 TO SIZEOF(AO_Word)/SIZEOF(AO_Word[0])-1 DO
		SlaveConfig.p_holding_registers[idx] := ADR(AO_Word[idx]);
	END_FOR;
	FOR idx:=0 TO SIZEOF(AI_Word)/SIZEOF(AI_Word[0])-1 DO
		SlaveConfig.p_input_registers[idx]	:= ADR(AI_Word[idx]);
	END_FOR;

	(* --------------------------------------------------------------------
	  Configure FUNCTION block instance
	  --------------------------------------------------------------------- *)
	ModbusTcpSlave.enable			:= 1; 					(* Enable function block *)
	ModbusTcpSlave.device			:= ADR('IF2');			(* Ethernet device string *)
	ModbusTcpSlave.p_cfg			:= ADR(SlaveConfig); 	(* IO configuration *)
	ModbusTcpSlave.master_timeout 	:= 5000; 				(* Disconnect master after x miliseconds when no request was sent, 0 = disabled *)

	(* The LOG information will show communication details. Enable for debugging,
	   disable FOR production TO save system resources *)
	ModbusTcpSlave.log.data_lines 	:= 20; 					(* Number of logging lines *)
	ModbusTcpSlave.log.pData 		:= ADR(logger);			(* Pointer to logger string array *)
	StartStop := 1;
END_PROGRAM

PROGRAM _CYCLIC
	(* --------------------------------------------------------------------
	  Cyclic FUNCTION call
	  --------------------------------------------------------------------- *)
	IF(StartStop) THEN
		ModbusTcpSlave();
	END_IF

	(* --------------------------------------------------------------------
	  Reset last error information
	  --------------------------------------------------------------------- *)
	IF(reset_error) THEN
		memset(ADR(ModbusTcpSlave.last_error), 0, 2);
		reset_error := 0;
	END_IF
END_PROGRAM
```

Listed in the project but not available here: Logical/CustomVars.var, Logical/Robo_Drive_Control/Robo_Drive.typ, Logical/Robo_Drive_Control/Robo_Drive.var, Logical/Robo_Drive_Control/FC302/FC302.typ, Logical/Robo_Drive_Control/FC302/FC302.var, Logical/Robo_Drive_Control/FC302/FC302.fun, Logical/Robo_Drive_Control/FC302/FC302_WriteParam.ab, Logical/Robo_Drive_Control/FC302/FC302_ReadSTW.ab, Logical/Robo_Drive_Control/FC302/FC302_WriteCTW.ab, Logical/Robo_Drive_Control/FC302/FC302_ReadParamTbl.ab, Logical/Robo_Drive_Control/FC302/FC302_ReadParam.ab, Logical/Robo_Drive_Control/zzRoboPosnNames/zzRoboPosnNames.ab, Logical/Robo_Drive_Control/zzRoboPosnNames/zzRoboPosnNames.typ, Logical/Robo_Drive_Control/zzRoboPosnNames/zzRoboPosnNames.var, Logical/Robo_Drive_Control/zzRoboPosnNamesTest/zzRoboPosnNamesTest.ab, Logical/Robo_Drive_Control/zzRoboPosnNamesTest/zzRoboPosnNamesTest.typ, Logical/Robo_Drive_Control/zzRoboPosnNamesTest/zzRoboPosnNamesTest.var, Logical/Robo_Drive_Control/Lift_PosMonitor, Logical/Robo_Drive_Control/31_vc1/vc.var, Logical/Robo_Drive_Control/31_vc1/vc.ab, Logical/Robo_Drive_Control/31_vc1/_httpRequest.st, Logical/Robo_Drive_Control/Lift_v8_1/Lift.var, Logical/Robo_Drive_Control/Lift_v8_1/Lift.ab, Logical/custom/HoistLibrary/Hoist.var, Logical/Rails, Logical/Device/Device_IDS.var, Logical/Device/Device.var, Logical/http_Lib/Request_Constants.var, Logical/http_Lib/Server_Functions.var, Logical/http_Lib/Constants.var, Logical/http_Lib/Variables.var, Logical/http_Lib/Types.typ, Logical/http_Lib/KanHttp/Types.typ, Logical/http_Lib/KanHttp/KanHttp.fun, Logical/http_Lib/KanHttp/httpGetParameter.st, Logical/http_Lib/zzHttpDriver/Types.typ, Logical/http_Lib/zzHttpDriver/Variables.var, Logical/http_Lib/zzHttpDriver/_ringBuffer.st, Logical/http_Lib/zzHttpDriver/_addToRing.st, Logical/http_Lib/zzHttpDriver/_orderRing.st, Logical/Bag1/Bag.var, Logical/Standard/Program, Logical/Standard/ABB_EPL/ABB_Driver/ControlWord.var, Logical/Standard/ABB_EPL/ABB_Driver/Types.typ, Logical/Standard/ABB_EPL/ABB_Driver/Variables.var, Logical/Standard/ABB_EPL/ABB_Driver/encodeParameters.st, Logical/Standard/ABB_EPL/ABB_Driver/_manual.st, Logical/Standard/ABB_EPL/ABB_Driver/_getNodeInfo.st, Logical/Standard/ABB_EPL/ABB_Driver/_packData.st, Logical/Standard/Barcode_BnR, Logical/Standard/Standard, Logical/Standard/HoistLibrary/Hoist.var, Logical/Standard/IOLink/Contactron/Contactron/Types.typ, Logical/Standard/IOLink/FuseManagement/Types.typ, Logical/Standard/Settings/Settings.var, Logical/Standard/Settings/Permenant/Variables.var, Logical/Standard/ToDO, Logical/Standard/Kanlink/Supertrack_Kanlink_Constants, Logical/Standard/Kanlink/KanLink_A19.typ, Logical/Standard/Kanlink/KanLink_A19.var, Logical/Standard/Kanlink/zz_KanlinkConfig/zz_KanlinkConfig.var, Logical/Standard/Kanlink/KGFramework/Pkg_KGStandard/Stat.var, Logical/Standard/Kanlink/KGFramework/Pkg_KGStandard/utfNames.typ, Logical/Standard/Kanlink/KGFramework/Pkg_KGStandard/kgbom.var, Logical/Standard/Kanlink/KGFramework/Pkg_KGStandard/KGstdLib/KG_Cmd.typ, Logical/Standard/Kanlink/KGFramework/Pkg_KGStandard/KGstdLib/Stat.typ, Logical/Standard/Kanlink/KGFramework/Pkg_KGStandard/KGstdLib/KGstdLib.typ, Logical/Standard/Kanlink/KGFramework/Pkg_KGStandard/KGstdLib/kgMachineState.typ, Logical/Standard/Kanlink/KGFramework/Pkg_KGStandard/KGstdLib/kgMachinetyp.typ, Logical/Standard/Kanlink/KGFramework/Pkg_KGStandard/KGstdLib/KG_Cmd.var, Logical/Standard/Kanlink/KGFramework/Pkg_KGStandard/KGstdLib/KGstdLib.var, Logical/Standard/Kanlink/KGFramework/Pkg_KGStandard/KGstdLib/kgMachineState.var, Logical/Standard/Kanlink/KGFramework/Pkg_KGStandard/KGstdLib/KGstdLib.fun, Logical/Standard/Kanlink/KGFramework/Pkg_KGStandard/KGstdLib/kgitoa_udint.st, Logical/Standard/Kanlink/KGFramework/Pkg_KGStandard/KGstdLib/kgatoi_udint.st, Logical/Standard/Kanlink/KGFramework/Pkg_KGStandard/KGstdLib/kgatoi_uint.st, Logical/Standard/Kanlink/KGFramework/Pkg_KGStandard/KGstdLib/kgInitBatchNoLong.st, Logical/Standard/Kanlink/KGFramework/Pkg_KGStandard/KGstdLib/kgNextBatchNoLong.st, Logical/Standard/Kanlink/KGFramework/Pkg_KGStandard/KGstdLib/kgGetMacAdress.st, Logical/Standard/Kanlink/KGFramework/Pkg_KGStandard/KGstdLib/kgGetBatchNoUnique.st, Logical/Standard/Kanlink/KGFramework/Pkg_KGStandard/KGstdLib/kgBatchNoToUDINT.st, Logical/Standard/Kanlink/KGFramework/Pkg_KGStandard/KGstdLib/kgUSINT16toGUID.st, Logical/Standard/Kanlink/KGFramework/Pkg_KGStandard/KGstdLib/kgGUIDtoSTRING.st, Logical/Standard/Kanlink/KGFramework/Pkg_KGStandard/KGstdLib/kgLogLine.st, Logical/Standard/Kanlink/KGFramework/Pkg_KGStandard/KGstdLib/kgArLogWrite.st, Logical/Standard/Kanlink/KGFramework/Pkg_KGStandard/KGstdLib/kgRBcreate.st, Logical/Standard/Kanlink/KGFramework/Pkg_KGStandard/KGstdLib/kgRBinsert.st, Logical/Standard/Kanlink/KGFramework/Pkg_KGStandard/KGstdLib/kgRBread.st, Logical/Standard/Kanlink/KGFramework/Pkg_KGStandard/KGstdLib/kgRBloc.st, Logical/Standard/Kanlink/KGFramework/Pkg_KGStandard/KGstdLib/kgGUIDisZero.st, Logical/Standard/Kanlink/KGFramework/Pkg_KGStandard/KGstdLib/kgRBbulkloc.st, Logical/Standard/Kanlink/KGFramework/Pkg_KGStandard/KGstdLib/kgGetLineNumberW3.st, Logical/Standard/Kanlink/KGFramework/Pkg_KGStandard/KGstdLib/kgGetMachineAdressW3.st, Logical/Standard/Kanlink/KGFramework/Pkg_KGStandard/KGstdLib/kgCheckDo.st, Logical/Standard/Kanlink/KGFramework/Pkg_KGStandard/KGstdLib/kgXOR.st, Logical/Standard/Kanlink/KGFramework/Pkg_KGStandard/KGstdLib/kgUnitconfREALtoDisplay.st, Logical/Standard/Kanlink/KGFramework/Pkg_KGStandard/KGstdLib/kgUnitconfDisplayToREAL.st, Logical/Standard/Kanlink/KGFramework/Pkg_KGStandard/KGstdLib/kgGetProgdata.st, Logical/Standard/Kanlink/KGFramework/Pkg_KGStandard/KGstdLib/kgSignalLight.st, Logical/Standard/Kanlink/KGFramework/Pkg_mnSystem/mnSystem/mnSystemCyclic.st, Logical/Standard/Kanlink/KGFramework/Pkg_mnSystem/mnSystem/mnSystemInit.st, Logical/Standard/Kanlink/KGFramework/Pkg_mnSystem/mnSystem/mnSystem.typ, Logical/Standard/Kanlink/KGFramework/Pkg_mnSystem/mnSystem/mnSystem.var, Logical/Standard/Kanlink/KGFramework/Pkg_mnSystem/Pkg_mnSystem.typ, Logical/Standard/Kanlink/KGFramework/Pkg_mnSystem/Pkg_mnSystem.var, Logical/Standard/Kanlink/KGFramework/Pkg_mnEth/Pkg_mnEth.typ, Logical/Standard/Kanlink/KGFramework/Pkg_mnEth/Pkg_mnEth.var, Logical/Standard/Kanlink/KGFramework/Pkg_mnEth/mnEth/mnEthCyclic.st, Logical/Standard/Kanlink/KGFramework/Pkg_mnEth/mnEth/mnEthInit.st, Logical/Standard/Kanlink/KGFramework/Pkg_mnEth/mnEth/mnEth.typ, Logical/Standard/Kanlink/KGFramework/Pkg_mnEth/mnEth/mnEth.var, Logical/Standard/Kanlink/KGFramework/Pkg_mnCnt/Pkg_mnCnt.typ, Logical/Standard/Kanlink/KGFramework/Pkg_mnCnt/Pkg_mnCnt.var, Logical/Standard/Kanlink/KGFramework/Pkg_mnCnt/mnCnt/mnCntCyclic.st, Logical/Standard/Kanlink/KGFramework/Pkg_mnCnt/mnCnt/mnCntInit.st, Logical/Standard/Kanlink/KGFramework/Pkg_mnCnt/mnCnt/mnCnt.typ, Logical/Standard/Kanlink/KGFramework/Pkg_mnCnt/mnCnt/mnCnt.var, Logical/Standard/Kanlink/KGFramework/Pkg_mnMsg/Pkg_mnMsg.typ, Logical/Standard/Kanlink/KGFramework/Pkg_mnMsg/Pkg_mnMsg.var, Logical/Standard/Kanlink/KGFramework/Pkg_mnMsg/mnMsg/mnMsgCyclic.st, Logical/Standard/Kanlink/KGFramework/Pkg_mnMsg/mnMsg/mnMsgInit.st, Logical/Standard/Kanlink/KGFramework/Pkg_mnMsg/mnMsg/mnMsg.typ, Logical/Standard/Kanlink/KGFramework/Pkg_mnMsg/mnMsg/mnMsg.var, Logical/Standard/Kanlink/KGFramework/Pkg_mnMsg/mnMsg/_actGetTxtFim.st, Logical/Standard/Kanlink/KGFramework/Pkg_mnMsg/mnMsg/_actGetTxtFimh.st, Logical/Standard/Kanlink/KGFramework/Pkg_mnMsg/mnMsg/_actGetOneTurnRB.st, Logical/Standard/Kanlink/KGFramework/Pkg_mnMsg/mnMsg/_actSetMsgOrMaint.st, Logical/Standard/Kanlink/KGFramework/Pkg_mnMsg/mnMsg/_actInsertRB.st, Logical/Standard/Kanlink/KGFramework/Pkg_mnMsg/mnMsg/_actInsertMsgL.st, Logical/Standard/Kanlink/KGFramework/Pkg_mnMsg/mnMsg/_actStatisticTextLCID.st, Logical/Standard/Kanlink/KGFramework/Pkg_mnMsg/mnMsg/_actLocMOD.st, Logical/Standard/Kanlink/KGFramework/Pkg_mnMsg/mnMsg/_actEventClassSel.st, Logical/Standard/Kanlink/KGFramework/Pkg_mnMsg/KGlibMsg/KGlibMsg.typ, Logical/Standard/Kanlink/KGFramework/Pkg_mnMsg/KGlibMsg/KGlibMsg.var, Logical/Standard/Kanlink/KGFramework/Pkg_mnMsg/KGlibMsg/KGlibMsg.fun, Logical/Standard/Kanlink/KGFramework/Pkg_mnMsg/KGlibMsg/msgBinSearchCfgList.st, Logical/Standard/Kanlink/KGFramework/Pkg_mnMsg/KGlibMsg/msgInsertMsgLine.st, Logical/Standard/Kanlink/KGFramework/Pkg_mnMsg/KGlibMsg/msgBinSearchTxtLine.st, Logical/Standard/Kanlink/KGFramework/Pkg_mnMsg/KGlibMsg/msgBinSearchHelpTxtLine.st, Logical/Standard/Kanlink/KGFramework/Pkg_mnMsg/KGlibMsg/msgReplSubStr.st, Logical/Standard/Kanlink/KGFramework/Pkg_mnMsg/KGlibMsg/msgNextChrPos.st, Logical/Standard/Kanlink/KGFramework/Pkg_mnParam/mnParam.typ, Logical/Standard/Kanlink/KGFramework/Pkg_mnParam/mnParam.var, Logical/Standard/Kanlink/KGFramework/Pkg_mnParam/mnParam/mnParamCyclic.st, Logical/Standard/Kanlink/KGFramework/Pkg_mnParam/mnParam/mnParamInit.st, Logical/Standard/Kanlink/KGFramework/Pkg_mnParam/mnParam/mnParamExit.st, Logical/Standard/Kanlink/KGFramework/Pkg_mnParam/mnParam/_mnParam.typ, Logical/Standard/Kanlink/KGFramework/Pkg_mnParam/mnParam/_mnParam.var, Logical/Standard/Kanlink/KGFramework/Pkg_mnParam/mnParam/_ExportContainer.st, Logical/Standard/Kanlink/KGFramework/Pkg_mnParam/mnParam/_ExportToc.st, Logical/Standard/Kanlink/KGFramework/Pkg_mnParam/mnParam/_DefActContainer.st, Logical/Standard/Kanlink/KGFramework/Pkg_mnParam/mnParam/_GetRights.st, Logical/Standard/Kanlink/KGFramework/Pkg_mnParam/mnParam/_BinSearchTxtLine.st, Logical/Standard/Kanlink/KGFramework/Pkg_mnParam/mnParam/_BinSearchHlpTxtLine.st, Logical/Standard/Kanlink/KGFramework/Pkg_mnParam/mnParam/_LimParam.st, Logical/Standard/Kanlink/KGFramework/Pkg_mnParam/mnParam/mnParam.fun, Logical/Standard/Kanlink/KGFramework/Pkg_mnParam/mnParam/_actInterfacePC.st, Logical/Standard/Kanlink/KGFramework/Pkg_mnParam/mnParam/_actInterfaceApplication.st, Logical/Standard/Kanlink/KGFramework/Pkg_mnParam/mnParam/_actFillEditNum.st, Logical/Standard/Kanlink/KGFramework/Pkg_mnParam/mnParam/_actFillEditStr.st, Logical/Standard/Kanlink/KGFramework/Pkg_mnParam/mnParam/_actFillNamelist.st, Logical/Standard/Kanlink/KGFramework/Pkg_mnParam/mnParam/_actImpModel.st, Logical/Standard/Kanlink/KGFramework/Pkg_mnParam/mnParamLib/mnParamLib.typ, Logical/Standard/Kanlink/KGFramework/Pkg_mnParam/mnParamLib/mnParamLib.var, Logical/Standard/Kanlink/KGFramework/Pkg_mnParam/mnParamLib/mnParamLib.fun, Logical/Standard/Kanlink/KGFramework/Pkg_mnParam/mnParamLib/mnParam_BinarySearchInNumeric.st, Logical/Standard/Kanlink/KGFramework/Pkg_mnParam/mnParamLib/mnParam_BinarySearchInString.st, Logical/Standard/Kanlink/KGFramework/Pkg_mnParam/mnParamLib/mnParam_CountLines.st, Logical/Standard/Kanlink/KGFramework/Pkg_mnParam/mnParamLib/mnParam_GetCsvDat.st, Logical/Standard/Kanlink/KGFramework/Pkg_mnParam/mnParamLib/mnParam_atodatetime.st, Logical/Standard/Kanlink/KGFramework/Pkg_mnParam/mnParamLib/mnParam_GetNextSubstring.st, Logical/Standard/Kanlink/KGFramework/Pkg_mnParam/mnParamLib/mnParam_GetContainerOfParamNum.st, Logical/Standard/Kanlink/KGFramework/Pkg_mnParam/mnParamLib/mnParam_GetContainerOfParamStrin.st, Logical/Standard/Kanlink/KGFramework/Pkg_mnParam/mnParamLib/GetArrayPV.st, Logical/Standard/Kanlink/KGFramework/Pkg_mnParam/mnParamLib/mnParam_WritePVNum.st, Logical/Standard/Kanlink/KGFramework/Pkg_mnParam/mnParamLib/mnParam_WritePVrNum.st, Logical/Standard/Kanlink/KGFramework/Pkg_mnParam/mnParamLib/mnParam_WritePVString.st, Logical/Standard/Kanlink/KGFramework/Pkg_mnParam/mnParamLib/mnParam_WriteBOM_Mem.st, Logical/Standard/Kanlink/KGFramework/Pkg_mnParam/mnParamLib/mnParam_WriteNewline_Mem.st, Logical/Standard/Kanlink/KGFramework/Pkg_mnParam/mnParamLib/mnParam_WriteCSV10_Mem.st, Logical/Standard/Kanlink/KGFramework/Pkg_mnParam/mnParamLib/mnParam_WriteCSV11_Mem.st, Logical/Standard/Kanlink/KGFramework/Pkg_mnParam/mnParamLib/mnParam_WriteCSV20_Mem.st, Logical/Standard/Kanlink/KGFramework/Pkg_mnParam/mnParamLib/mnParam_WriteCSV81_Mem.st, Logical/Standard/Kanlink/KGFramework/Pkg_mnParam/mnParamLib/mnParam_WriteCSV80_Mem.st, Logical/Standard/Kanlink/KGFramework/Pkg_mnParam/mnParamLib/mnParam_WriteCSV90_Mem.st, Logical/Standard/Kanlink/KGFramework/Pkg_mnParam/mnParamLib/mnParam_WriteCSV251_Mem.st, Logical/Standard/Kanlink/KGFramework/Pkg_mnParam/mnParamLib/mnParam_WriteCSV252_Mem.st, Logical/Standard/Kanlink/KGFramework/Pkg_mnParam/mnParamLib/mnParam_WriteCSV253_Mem.st, Logical/Standard/Kanlink/KGFramework/Pkg_mnParam/mnParamLib/mnParam_WriteCSV254_Mem.st, Logical/Standard/Kanlink/KGFramework/Pkg_mnParam/mnParamLib/mnParam_WriteCSV255_Mem.st, Logical/Standard/Kanlink/KGFramework/Pkg_mnParam/mnParamLib/mnParam_datetimetoa.st, Logical/Standard/Kanlink/KGFramework/Pkg_mnParam/mnParamLib/mnParam_datetoa.st, Logical/Standard/Kanlink/KGFramework/Pkg_mnTxt/Pkg_mnTxt.typ, Logical/Standard/Kanlink/KGFramework/Pkg_mnTxt/Pkg_mnTxt.var, Logical/Standard/Kanlink/KGFramework/Pkg_mnTxt/mnTxt/mnTxtCyclic.st, Logical/Standard/Kanlink/KGFramework/Pkg_mnTxt/mnTxt/mnTxtInit.st, Logical/Standard/Kanlink/KGFramework/Pkg_mnTxt/mnTxt/mnTxt.typ, Logical/Standard/Kanlink/KGFramework/Pkg_mnTxt/mnTxt/mnTxt.var, Logical/Standard/Kanlink/KGFramework/Pkg_mnTxt/mnTxt/_utfReplaceCtrl.st, Logical/Standard/Kanlink/KGFramework/Pkg_mnTxt/mnTxt/mnTxt.fun, Logical/Standard/Kanlink/KGFramework/Pkg_hlDFII/Pkg_hlDFII.typ, Logical/Standard/Kanlink/KGFramework/Pkg_hlDFII/Pkg_hlDFII.var, Logical/Standard/Kanlink/KGFramework/Pkg_hlDFII/hlDFII/hlDFIICyclic.st, Logical/Standard/Kanlink/KGFramework/Pkg_hlDFII/hlDFII/hlDFIIInit.st, Logical/Standard/Kanlink/KGFramework/Pkg_hlDFII/hlDFII/hlDFIIExit.st, Logical/Standard/Kanlink/KGFramework/Pkg_hlDFII/hlDFII/hlDFII.typ, Logical/Standard/Kanlink/KGFramework/Pkg_hlDFII/hlDFII/hlDFII.var, Logical/Standard/Kanlink/KGFramework/Pkg_hlDFII/hlDFII/_actReqScheduleTrack.st, Logical/Standard/Kanlink/KGFramework/Pkg_hlDFII/hlDFII/_actReqScheduleDFII.st, Logical/Standard/Kanlink/KGFramework/Pkg_hlDFII/hlDFII/_actProcCmdTrack.st, Logical/Standard/Kanlink/KGFramework/Pkg_hlDFII/hlDFII/_actProcCmdDFII.st, Logical/Standard/Kanlink/KGFramework/Pkg_hlDFII/hlDFII/_actProcSQLTrack.st, Logical/Standard/Kanlink/KGFramework/Pkg_hlDFII/hlDFII/_actProcSQLDFII.st, Logical/Standard/Kanlink/KGFramework/Pkg_hlDFII/hlDFII/_CreateConnectionString.st, Logical/Standard/Kanlink/KGFramework/Pkg_hlDFII/hlDFII/hlDFII.fun, Logical/Standard/Kanlink/KGFramework/Pkg_mnTest/Pkg_mnTest.typ, Logical/Standard/Kanlink/KGFramework/Pkg_mnTest/Pkg_mnTest.var, Logical/Standard/Kanlink/KGFramework/Pkg_mnTest/mnTest/mnTestCyclic.st, Logical/Standard/Kanlink/KGFramework/Pkg_mnTest/mnTest/mnTestInit.st, Logical/Standard/Kanlink/KGFramework/Pkg_mnTest/mnTest/mnTestExit.st, Logical/Standard/Kanlink/KGFramework/Pkg_mnTest/mnTest/mnTest.typ, Logical/Standard/Kanlink/KGFramework/Pkg_mnTest/mnTest/mnTest.var, Logical/Standard/Kanlink/KGFramework/Pkg_mnTest/mnTest/_MessageTest1.st, Logical/Standard/Kanlink/KGFramework/Pkg_svCPCache/Pkg_svCPCache.typ, Logical/Standard/Kanlink/KGFramework/Pkg_svCPCache/Pkg_svCPCache.var, Logical/Standard/Kanlink/KGFramework/Pkg_svCPCache/svCPCache/svCPCacheCyclic.st, Logical/Standard/Kanlink/KGFramework/Pkg_svCPCache/svCPCache/svCPCacheInit.st, Logical/Standard/Kanlink/KGFramework/Pkg_svCPCache/svCPCache/svCPCacheExit.st, Logical/Standard/Kanlink/KGFramework/Pkg_svCPCache/svCPCache/svCPCache.typ, Logical/Standard/Kanlink/KGFramework/Pkg_svCPCache/svCPCache/svCPCache.var, Logical/Standard/Kanlink/KGFramework/Pkg_svCPCache/svCPCache/_actCPImport.st, Logical/Standard/Kanlink/KGFramework/Pkg_svCPCache/svCPCache/_actIFCmd.st, Logical/Standard/Kanlink/KGFramework/Pkg_svCPCache/svCPCache/_actFillCPList.st, Logical/Standard/Kanlink/KGFramework/Pkg_svCPCache/svCPCache/_actSaveCSV.st, Logical/Standard/Kanlink/KGFramework/Pkg_svCPCache/svCPCache/_TrimCategory.st, Logical/Standard/Kanlink/KGFramework/Pkg_svCPCache/svCPCache/svCPCache.fun, Logical/Standard/Kanlink/KGFramework/Pkg_hlKanLink/hlKanLink.typ, Logical/Standard/Kanlink/KGFramework/Pkg_hlKanLink/hlKanLink.var, Logical/Standard/Kanlink/KGFramework/Pkg_hlKanLink/hlKanLink/KanLink.typ, Logical/Standard/Kanlink/KGFramework/Pkg_hlKanLink/hlKanLink/KanLink.var, Logical/Standard/Kanlink/KGFramework/Pkg_hlKanLink/hlKanLink/KanLinkInit.st, Logical/Standard/Kanlink/KGFramework/Pkg_hlKanLink/hlKanLink/KL_SaveConfDO.st, Logical/Standard/Kanlink/KGFramework/Pkg_hlKanLink/hlKanLink/KanLink.fun, Logical/Standard/Kanlink/KGFramework/Pkg_hlKanLink/hlKanLink/actGetServerReq.st, Logical/Standard/Kanlink/KGFramework/Pkg_hlKanLink/hlKanLink/actResponse.st, Logical/Standard/Kanlink/KGFramework/Pkg_hlKanLink/KanLinkLib/CmdBTxfer.typ, Logical/Standard/Kanlink/KGFramework/Pkg_hlKanLink/KanLinkLib/CmdBI.typ, Logical/Standard/Kanlink/KGFramework/Pkg_hlKanLink/KanLinkLib/CmdSI.typ, Logical/Standard/Kanlink/KGFramework/Pkg_hlKanLink/KanLinkLib/CmdSilo.typ, Logical/Standard/Kanlink/KGFramework/Pkg_hlKanLink/KanLinkLib/KLInterface.typ, Logical/Standard/Kanlink/KGFramework/Pkg_hlKanLink/KanLinkLib/KanLinkLib.typ, Logical/Standard/Kanlink/KGFramework/Pkg_hlKanLink/KanLinkLib/KanLinkLib.var, Logical/Standard/Kanlink/KGFramework/Pkg_hlKanLink/KanLinkLib/KanLinkLib.fun, Logical/Standard/Kanlink/KGFramework/Pkg_hlKanLink/KanLinkLib/KLLib_CfgClient.st, Logical/Standard/Kanlink/KGFramework/Pkg_hlKanLink/KanLinkLib/KLLib_CfgServer.st, Logical/Standard/Kanlink/KGFramework/Pkg_hlKanLink/KanLinkLib/KanLink_FB.st, Logical/Standard/Kanlink/KGFramework/Pkg_hlKanLink/KanLinkLib/KLLib_ClientTimer.st, Logical/Standard/Kanlink/KGFramework/Pkg_hlKanLink/KanLinkLib/KLLib_GetPVAdr.st, Logical/Standard/Kanlink/KGFramework/Pkg_hlKanLink/KanLinkLib/KLLib_SendData.st, Logical/Standard/Kanlink/KGFramework/Pkg_hlKanLink/KanLinkLib/KLLib_ReadServerPara.st, Logical/Standard/Kanlink/KGFramework/Pkg_hlKanLink/KanLinkLib/KLLib_InitCltPV.st, Logical/Standard/Kanlink/KGFramework/Pkg_hlKanLink/KanLinkLib/KLLib_ReadClientPara.st, Logical/Standard/Kanlink/KGFramework/Pkg_hlKanLink/KanLinkLib/KL_BuildKey.st, Logical/Standard/Kanlink/KGFramework/Pkg_hlKanLink/KanLinkLib/KLLib_Init.st, Logical/Standard/Kanlink/KGFramework/Pkg_hlKanLink/KanLinkLib/KLLib_CreateStrucDef.st, Logical/Standard/Kanlink/KGFramework/Pkg_hlKanLink/KanLinkLib/KLLib_WriteStrucDefLine.st, Logical/Standard/Kanlink/KGFrameworkShare/hlDFII.Glob.var, Logical/Standard/Kanlink/KGFrameworkShare/mnCntGlob.var, Logical/Standard/Kanlink/KGFrameworkShare/mnTxtGlob.var, Logical/Standard/Kanlink/KGFrameworkShare/mnParamGlob.var, Logical/Standard/Kanlink/KGFrameworkShare/svCPCacheGlob.var, Logical/Standard/Kanlink/KGFrameworkShare/mnSystemGlob.var, Logical/Standard/Kanlink/KGFrameworkShare/Pkg_KGStandardShare/KGStandardShare.kgMsgStatus.var, Logical/Standard/Kanlink/KGFrameworkShare/Pkg_KGStandardShare/kgdevice.var, Logical/Standard/Kanlink/KGFrameworkShare/Pkg_mnEthShare/Pkg_mnEthShare.var, Logical/Standard/Kanlink/KGFrameworkShare/Pkg_mnMsgShare/Pkg_mnMsgShare.var, Logical/Standard/Kanlink/KGFrameworkShare/Pkg_hlKanLinkUser/Pkg_hlKanLinkUser.var, Logical/Standard/Kanlink/KGFrameworkShare/Pkg_hlKanLinkUser/KL_UserLib/Batch.typ, Logical/Standard/Kanlink/KGFrameworkShare/Pkg_hlKanLinkUser/KL_UserLib/KL_UserLib.typ, Logical/Standard/Kanlink/KGFrameworkShare/Pkg_hlKanLinkUser/KL_UserLib/KL_OnRecReq.st, Logical/Standard/Kanlink/KGFrameworkShare/Pkg_hlKanLinkUser/KL_UserLib/KL_UserLib.fun, Logical/Standard/Kanlink/KGFrameworkShare/Pkg_hlKanLinkUser/KL_UserLib/CmdWetExt.typ, Logical/Standard/Kanlink/KGFrameworkShare/Pkg_mnTestUser/libTestUse/libTest.typ, Logical/Standard/Kanlink/KGFrameworkShare/Pkg_mnTestUser/libTestUse/libTestUse.typ, Logical/Standard/Kanlink/KGFrameworkShare/Pkg_mnTestUser/libTestUse/libTest.var, Logical/Standard/Kanlink/KGFrameworkShare/Pkg_mnTestUser/libTestUse/libTestUse.var, Logical/Standard/Kanlink/KGFrameworkShare/Pkg_mnTestUser/libTestUse/TestUser_StopTask.st, Logical/Standard/Kanlink/KGFrameworkShare/Pkg_mnTestUser/libTestUse/TestUser_SetMode.st, Logical/Standard/Kanlink/KGFrameworkShare/Pkg_mnTestUser/libTestUse/TestUser_RunTest.st, Logical/Standard/Kanlink/KGFrameworkShare/Pkg_mnTestUser/libTestUse/libTestUse.fun, Logical/Standard/Kanlink/KGFrameworkShare/Pkg_mnTestUser/mnTestUser/mnTestUserCyclic.st, Logical/Standard/Kanlink/KGFrameworkShare/Pkg_mnTestUser/mnTestUser/mnTestUserInit.st, Logical/Standard/Kanlink/KGFrameworkShare/Pkg_mnTestUser/mnTestUser/mnTestUserExit.st, Logical/Standard/Kanlink/KGFrameworkShare/Pkg_mnTestUser/mnTestUser/mnTestUser.typ, Logical/Standard/Kanlink/KGFrameworkShare/Pkg_mnTestUser/mnTestUser/mnTestUser.var, Logical/Standard/Safety/Safety.typ, Logical/Standard/Safety/Safety.var, Logical/Standard/Safety/mappSafety.var, Logical/Standard/Safety/mappSafety.typ, Logical/Standard/Safety/mappSafety/Main.st, Logical/Standard/Safety/mappSafety/Types.typ, Logical/Standard/Safety/mappSafety/Variables.var, Logical/Standard/Safety/EvueSafety/Types.typ, Logical/Standard/Safety/EvueSafety/Variables.var, Logical/Standard/Safety/EvueSafety/_decodeData.st, Logical/Standard/Safety/SafetyUI/SafetyUI.typ, Logical/Standard/Safety/SafetyUI/SafetyUI.fun, Logical/Standard/Safety/SafetyUI/itoahex.st, Logical/COMMUNICATION/Communication.typ, Logical/COMMUNICATION/MbusTCP/MbusTCP.fun, Logical/COMMUNICATION/MbusTCP/MbusTCP.typ, Logical/COMMUNICATION/MbusTCP/MBmaster.c, Logical/COMMUNICATION/MbusTCP/MBslave.c, Logical/COMMUNICATION/MbusTCP/MBcommon.c, Logical/COMMUNICATION/MbusTCP/MBdeclarations.h, Logical/COMMUNICATION/ModSlave/ModSlave.var, Logical/COMMUNICATION/tcpComm/Types.typ, Logical/COMMUNICATION/tcpComm/Variables.var, Logical/COMMUNICATION/tcpComm/Responses.var, Logical/COMMUNICATION/tcpComm/_references.st, Logical/COMMUNICATION/tcpComm/_decodeModbus.st, Logical/COMMUNICATION/tcpComm/_messageAcknowledge.st, Logical/Bag/http_Lib/Request_Constants.var, Logical/Bag/http_Lib/Server_Functions.var, Logical/Bag/http_Lib/Constants.var, Logical/Bag/http_Lib/Variables.var, Logical/Bag/http_Lib/httpServer/_vcCommand.st, Logical/Bag/http_Lib/httpServer/_apiFunctions.st, Logical/Bag/http_Lib/httpServer/_getFunctionName.st, Logical/Bag/http_Lib/httpServer/_setBagDestination.st, Logical/Bag/http_Lib/httpServer/_setBeltConfig.st, Logical/Bag/http_Lib/httpServer/_getLoadingData.st, Logical/Bag/http_Lib/httpServer/_PostAbbManual.st, Logical/Bag/http_Lib/httpServer/_httpServer.st, Logical/Bag/http_Lib/httpServer/Types.typ, Logical/Bag/http_Lib/httpServer/LocalFunctions.fun, Logical/Bag/http_Lib/httpServer/httpGetParameter.st, Logical/Bag/http_Lib/zzHttpDriver, Logical/IOLink/IOLink_Driver/Types.typ, Logical/IOLink/IOLink_Driver/Variables.var, Logical/IOLink/IOLink_Driver/_EasyB.st, Logical/IOLink/IOLink_Driver/_status.st, Logical/IOLink/IOLink_Driver/backUpWrite.st, Logical/IOLink/IOLink_Driver/backUpRead.st, Logical/IOLink/IOLink_Driver/encodeData.st, Logical/IOLink/IOLink_Driver/decodeData.st, Logical/IOLink/FuseManagement/Constants.var, Logical/IOLink/IOLinkLib/Types.typ, Logical/IOLink/IOLinkLib/IOLinkLib.fun
